// TIA Portal V18 export
FUNCTION "WeekScheduler" : Void   // FC98, LAD
{ S7_Optimized_Access := 'TRUE' }
VERSION : 0.1
// stored: AutoNumber false, IsIECCheckEnabled false, SetENOAutomatically false, UDAEnableTagReadback false
   VAR_INPUT
      Mon_PreComfort_Start : Time_Of_Day;
      Mon_PreComfort_Stop : Time_Of_Day;
      Mon_Comfort_Start : Time_Of_Day;
      Mon_Comfort_Stop : Time_Of_Day;
      WD_PreComfort_Start : Time_Of_Day;
      WD_PreComfort_Stop : Time_Of_Day;
      WD_Comfort_Start : Time_Of_Day;
      WD_Comfort_Stop : Time_Of_Day;
      Sat_PreComfort_Start : Time_Of_Day;
      Sat_PreComfort_Stop : Time_Of_Day;
      Sat_Comfort_Start : Time_Of_Day;
      Sat_Comfort_Stop : Time_Of_Day;
      Sun_PreComfort_Start : Time_Of_Day;
      Sun_PreComfort_Stop : Time_Of_Day;
      Sun_Comfort_Start : Time_Of_Day;
      Sun_Comfort_Stop : Time_Of_Day;
      Hol_PreComfort_Start : Time_Of_Day;
      Hol_PreComfort_Stop : Time_Of_Day;
      Hol_Comfort_Start : Time_Of_Day;
      Hol_Comfort_Stop : Time_Of_Day;
      Holidays : Array[1..4] of Date;
   END_VAR
   VAR_OUTPUT
      cOpModeNow : Byte;
      xIsHoliday : Bool;
      cDayType : Byte;   // 1-WD/2-Sat/3-Sun/4 - Hol
      CurrentDate : Date;
      CurrentTOD : Time_Of_Day;
      iRetVal : Int;
   END_VAR
   VAR_TEMP
      NowDTL : DTL;
      i : Int;
      PreComfStart : Time_Of_Day;
      PreComfStop : Time_Of_Day;
      ComfStart : Time_Of_Day;
      ComfStop : Time_Of_Day;
      xInPreComf : Bool;
      xInComf : Bool;
   END_VAR
BEGIN

REGION Network 1 (SCL): // Значення за замовчуванням
       // Значення за замовчуванням
      // #cOpModeNow := 1; // Економ
      // #xIsHoliday := FALSE;
      // #cDayType := 1; // Робочий
      // #CurrentDate := DATE#1990-01-01;
      // #CurrentTOD := TOD#00:00:00;
      // #iRetVal := 0;
END_REGION

REGION Network 2 (SCL): Час на CPU
   // Читаємо локальний час CPU
   #iRetVal := RD_LOC_T(OUT => #NowDTL);

   // Якщо час не прочитався - лишаємо Економ
   //IF #iRetVal >= 16#8000 THEN
   //    #cOpModeNow := 1;
   //    RETURN;
   //END_IF;

   // Виділяємо дату і час
   #CurrentDate := DTL_TO_DATE(#NowDTL);
   #CurrentTOD := DTL_TO_TOD(#NowDTL);
END_REGION

REGION Network 3 (SCL): // Перевірка святкового дня
   // Перевірка святкового дня
   FOR #i := 1 TO 3 DO
       IF #Holidays[#i] = #CurrentDate THEN
           #xIsHoliday := TRUE;
           EXIT;
       END_IF;
   END_FOR;
END_REGION

REGION Network 4 (SCL): 0-WD/1-Mon/2-Sat/3-Sun/4 - Hol
       // Визначення типу дня
       IF #xIsHoliday THEN
           #cDayType := 4; // Святковий
       ELSE
           // Weekday: 1=Sunday ... 7=Saturday
           CASE #NowDTL.WEEKDAY OF
               7:
                   #cDayType := 2; // Субота
               1:
                   #cDayType := 3; // Неділя
               2:
                   #cDayType := 1; // Понеділок
               ELSE
                   #cDayType := 0; // Робочий
           END_CASE;
       END_IF;
END_REGION

REGION Network 5 (SCL): // Вибір активного розкладу
   // Вибір активного розкладу
   CASE #cDayType OF
       0: // Робочий
           #PreComfStart := #WD_PreComfort_Start;
           #PreComfStop := #WD_PreComfort_Stop;
           #ComfStart := #WD_Comfort_Start;
           #ComfStop := #WD_Comfort_Stop;

       1: // Понеділок
           #PreComfStart := #Mon_PreComfort_Start;
           #PreComfStop := #Mon_PreComfort_Stop;
           #ComfStart := #Mon_Comfort_Start;
           #ComfStop := #Mon_Comfort_Stop;

       2: // Субота
           #PreComfStart := #Sat_PreComfort_Start;
           #PreComfStop := #Sat_PreComfort_Stop;
           #ComfStart := #Sat_Comfort_Start;
           #ComfStop := #Sat_Comfort_Stop;

       3: // Неділя
           #PreComfStart := #Sun_PreComfort_Start;
           #PreComfStop := #Sun_PreComfort_Stop;
           #ComfStart := #Sun_Comfort_Start;
           #ComfStop := #Sun_Comfort_Stop;

       4: // Святковий
           #PreComfStart := #Hol_PreComfort_Start;
           #PreComfStop := #Hol_PreComfort_Stop;
           #ComfStart := #Hol_Comfort_Start;
           #ComfStop := #Hol_Comfort_Stop;

       ELSE
           #PreComfStart := TOD#00:00:00;
           #PreComfStop := TOD#00:00:00;
           #ComfStart := TOD#00:00:00;
           #ComfStop := TOD#00:00:00;

   END_CASE;
END_REGION

REGION Network 6 (SCL): // Перевірка потрапляння в інтервали InComf
       IF #ComfStart = #ComfStop THEN
           // трактуємо як "вікно вимкнене"
           #xInComf := FALSE;

       ELSIF #ComfStart <  #ComfStop THEN
           // звичайний інтервал, наприклад 06:00..22:00
           #xInComf := (#CurrentTOD >= #ComfStart) AND (#CurrentTOD < #ComfStop);

       ELSE
           // інтервал через північ, наприклад 22:00..06:00
           //#xInComf := (#CurrentTOD >= #ComfStart) OR (#CurrentTOD < #ComfStop);
           #xInComf := FALSE;
       END_IF;
END_REGION

REGION Network 7 (SCL): // Перевірка потрапляння в інтервали InPreComf
       IF #PreComfStart = #PreComfStop THEN
           // трактуємо як "вікно вимкнене"
           #xInPreComf := FALSE;

       ELSIF #PreComfStart < #PreComfStop THEN
           // звичайний інтервал, наприклад 06:00..22:00
           #xInPreComf := (#CurrentTOD >= #PreComfStart) AND (#CurrentTOD < #PreComfStop);

       ELSE
           // інтервал через північ, наприклад 22:00..06:00
           //#xInComf := (#CurrentTOD >= #ComfStart) OR (#CurrentTOD < #ComfStop);
           #xInPreComf := FALSE;
       END_IF;
END_REGION

REGION Network 8 (SCL): // Пріоритет: Комфорт > Прекомфорт > Економ
       // Пріоритет: Комфорт > Прекомфорт > Економ
       IF #xInComf THEN
           #cOpModeNow := 3; // Комфорт
       ELSIF #xInPreComf THEN
           #cOpModeNow := 2; // Прекомфорт
       ELSE
           #cOpModeNow := 1; // Економ
       END_IF;
END_REGION
END_FUNCTION
